{attribute 'linkalways'} 
{attribute 'no_explicit_call' := 'This FB is a CLASS and must be accessed using methods or properties'}
{attribute 'enable_dynamic_creation'}
FUNCTION_BLOCK Node_ContainerType_Vector_TcVnVector2_UINT EXTENDS Node
VAR
    out : _GUID;
END_VAR

METHOD PUBLIC  Clone : I_Node
VAR
	pNode : POINTER TO Node_ContainerType_Vector_TcVnVector2_UINT;
END_VAR
pNode := __NEW(Node_ContainerType_Vector_TcVnVector2_UINT);
Clone := pNode^;
END_METHOD

METHOD FB_init : BOOL
VAR_INPUT
	bInitRetains : BOOL; // if TRUE, the retain variables are initialized (warm start / cold start)
	bInCopyCode : BOOL;  // if TRUE, the instance afterwards gets moved into the copy code (online change)
END_VAR
AddOutput('out', out);
END_METHOD

METHOD PROTECTED OnExecute
out.Value := ContainerType_Vector_TcVnVector2_UINT;
END_METHOD

END_FUNCTION_BLOCK

(* stored: Version 1.1.0.1, ProductVersion 3.1.4026.17
   POU Node_ContainerType_Vector_TcVnVector2_UINT: Id {2a9f2ce2-6cc7-0349-11db-6d18d8419268}, SpecialFunc None
   Folder Constructor: Id {4b5cb5f3-2191-01ab-0882-b658bcea0b86}
   Method Clone: Id {0486c599-b167-067a-0f57-70a6e8ce7fce}
   Method FB_init: Id {ce124da0-0533-0296-29ff-f50c97c87ef7}
   Method OnExecute: Id {cade4b01-9918-0530-168b-06532582823f} *)
